# EPICS autosave request: 3-3/GalilSup/Db/galil_kinematic_variable.req
# Kinematic variables
$(P)$(R)_SP.VAL
